# EPICS substitutions: test/integrationTests/volumes/test/I34/volumes/bin/sourceIoc/sourceApp/Db/poz.substitutions
file db/test.template {
    pattern { N }
        { 1 }
        { 2 }
        { 3 }
        { 4 }
        { 5 }
}
